FUNCTION_BLOCK fbLoadMoves
VAR_INPUT
	DeltaCoords:Coords;
END_VAR
VAR_OUTPUT
END_VAR
VAR
END_VAR

END_FUNCTION_BLOCK

(* stored: Version 1.1.0.1, ProductVersion 3.1.4024.11
   POU fbLoadMoves: Id {fdf544d3-cc44-4532-b0ef-2d4f8a6412bc}, SpecialFunc None *)
